FUNCTION_BLOCK PUBLIC T_Enable IMPLEMENTS I_Enable
VAR
	axRef : REFERENCE TO AXIS_REF;
	_power : MC_Power;
	_busy : BOOL;
END_VAR

IF NOT __ISVALIDREF(axRef) THEN
	RETURN;
END_IF

_power(Axis := axRef);

PROPERTY Busy : bool
GET
Busy := _busy;
END_GET
END_PROPERTY

METHOD Disable : BOOL
VAR_INPUT
END_VAR
_power.Enable := false;
END_METHOD

METHOD Enable : BOOL
VAR_INPUT
END_VAR
_power.Enable := true;
END_METHOD

PROPERTY PUBLIC Error : bool
GET
Error := _power.Error OR NOT __ISVALIDREF(axRef)
END_GET
END_PROPERTY

METHOD PUBLIC Parameterise : BOOL
VAR_INPUT
	override : LREAL;
	enablePositive : BOOL;
	enableNegative : BOOL;
END_VAR
IF Busy THEN
	RETURN;
END_IF

_power.Override := override;
_power.Enable_Negative := enableNegative;
_power.Enable_Positive := enablePositive;

Parameterise := true;
END_METHOD

METHOD PUBLIC RegisterAxis : BOOL
VAR_IN_OUT
	axisRef : AXIS_REF;
END_VAR
IF Busy THEN
	RETURN;
END_IF
axRef REF=	axisRef;

RegisterAxis := true;
END_METHOD

END_FUNCTION_BLOCK

(* stored: Version 1.1.0.1, ProductVersion 3.1.4024.3
   POU T_Enable: Id {73c8894a-9971-4c06-882a-bfe6e428e44d}, SpecialFunc None
   Property Busy: Id {373d9411-fe86-4b98-8012-9ce31029fdc5}
   Get Get: Id {88e7bc56-0d60-4bdf-911b-f67de91427db}
   Method Disable: Id {7521d3dd-ee87-4851-8f1e-3bdcf4457226}
   Method Enable: Id {eb8294f5-8810-4584-b2b7-40295e78a6f1}
   Property Error: Id {0ee63d32-bb49-4fc5-907a-f201d8797441}
   Get Get: Id {234676ec-7c08-444e-8d06-b4578fb9880c}
   Method Parameterise: Id {cab59032-c731-4755-9942-acfc42775c4d}
   Method RegisterAxis: Id {a868cf8a-2d4d-4401-bd0c-1bfe9d59e3eb} *)
